TYPE ST_Chamber1SpinAxisMoveVelParam :
STRUCT
	Velocity : LREAL;
	Acceleration : LREAL;
	Deceleration : LREAL;
END_STRUCT
END_TYPE

(* stored: Version 1.1.0.1, ProductVersion 3.1.4026.18
   DUT ST_Chamber1SpinAxisMoveVelParam: Id {d1d16288-69ff-4d7a-a63b-4aedf7614d0b} *)
